FUNCTION proj3_TupleStruct_1: REAL
{ S7_Optimized_Access := 'false' }
    VAR_INPUT
        tuple: TupleStruct_1;
    END_VAR

BEGIN
    proj3_TupleStruct_1 := tuple.field3;
END_FUNCTION
